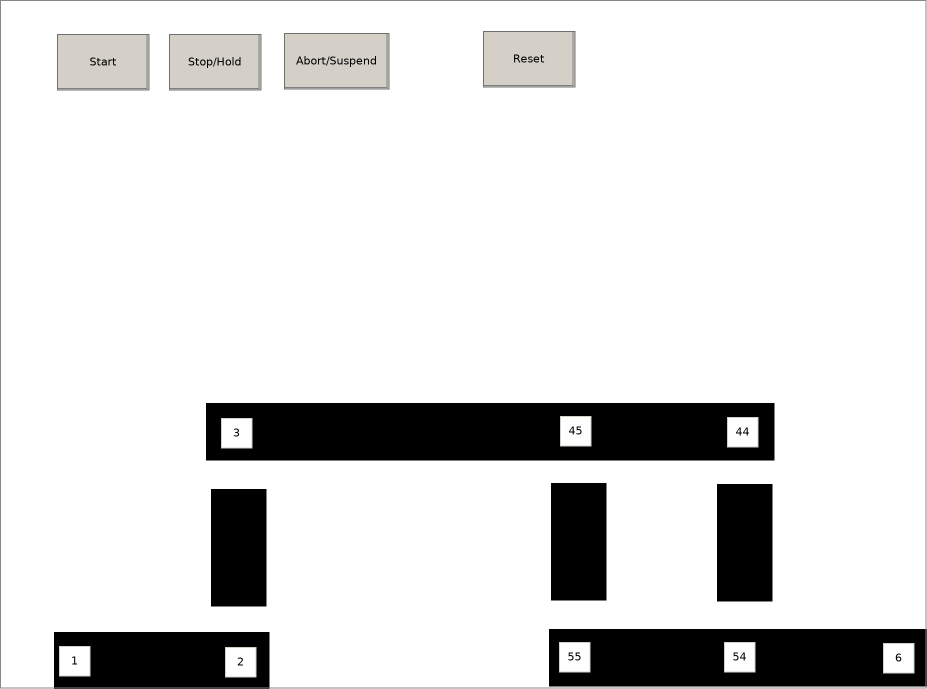
VISUALIZATION Visualization  // 927x689
    Rectangle (54,632 215x57)
    Button (57,34 92x56), "Start"
    Button (169,34 92x56), "Stop/Hold"
    Button (284,33 105x56), "Abort/Suspend"
    Button (483,31 92x56), "Reset"
    Rectangle (206,403 568x57)
    Rectangle (549,629 378x57)
    RoundedRectangle (211,489 55x117)
    RoundedRectangle (717,484 55x117)
    Textfield (59,646 31x30), "1"
    Textfield (225,647 31x30), "2"
    Textfield (221,418 31x30), "3"
    RoundedRectangle (551,483 55x117)
    Textfield (560,416 31x30), "45"
    Textfield (727,417 31x30), "44"
    Textfield (559,642 31x30), "55"
    Textfield (724,642 31x30), "54"
    Textfield (883,643 31x30), "6"
END_VISUALIZATION

(* stored: Version 1.1.0.1, ProductVersion 3.1.4024.12
   Visu Visualization: Id {07feb572-807c-455d-a2fd-a7a81f46326b} *)
